--- Up24.dat ---
&ACCESS RVO1
&REL 1255
&COMMENT VW380 Klebeauftrag_AFO415600
&PARAM EDITMASK = Up999[1-999]
&PARAM TEMPLATE = C:\KRC\Roboter\Template\upvorgabe
&PARAM TPVW_VERSION = 8.3.18
&PARAM DISKPATH = KRC:\R1\UPs
DEFDAT UP24
; FOLD ;%{H} %MKUKATPVW
; ENDFOLD
; interface to basic routines
 EXT  BAS (BAS_COMMAND  :IN,REAL  :IN )
; interface to VW-standard routines
EXT VW (VW_COMMAND:IN, BOOL: IN, REAL:IN, REAL:IN, REAL:IN, REAL:IN, BOOL :IN, E6POS :IN )
; interface to VW_USER - Call
EXT  VW_USER (VW_USER_CMD :IN,INT :IN,REAL  :IN,REAL  :IN,REAL  :IN,REAL  :IN,REAL  :IN,REAL  :IN,REAL  :IN,REAL  :IN,REAL  :IN,BOOL  :IN)
EXT  VW_USR_R (VW_USER_CMD :IN,INT :IN,REAL  :IN,REAL  :IN,REAL  :IN,REAL  :IN,REAL  :IN,REAL  :IN,REAL  :IN,REAL  :IN,REAL  :IN,BOOL  :IN)
EXT  IBGN (IBGN_COMMAND  :IN,BOOL  :IN,REAL  :IN,REAL  :IN,BOOL  :IN,E6POS  :OUT )
; interface select routine
EXTFCT INT  SELECT (SUBTYPE  :IN,INT  :IN,BOOL  :IN,ARI_TYP  :IN,INT  :IN,BOOL_TYP  :IN,INT  :IN,BOOL  :IN)
INT VW_NEXT_FREE = 145
INT VW_NFREE_SPS = 147
INT VW_MAX_SPS = 247
DECL VW_MPARA_TYP P1_D = {TOOL_NO 1,BASE_NO 2,VB 100,VE 0,ACC 100,TRG_TIME 0,MOVE_TYPE #PTP_MOTION}
DECL E6POS P1 = {X 1079.993, Y 23.2307, Z -59.63425, A -156.517, B 2.823335, C 116.2772, S 2, T 2 , E1 0.0, E2 0.0, E3 0.0, E4 0.0, E5 0.0, E6 0.0}
DECL VW_MPARA_TYP P2_D = {TOOL_NO 1,BASE_NO 2,VB 100,VE 100,ACC 100,TRG_TIME 0,MOVE_TYPE #PTP_MOTION}
DECL E6POS P2 = {X 1309.031, Y -94.76365, Z 183.6622, A -143.6638, B -5.59984, C 155.4084, S 2, T 2 , E1 0.0, E2 0.0, E3 0.0, E4 0.0, E5 0.0, E6 0.0}
DECL VW_MPARA_TYP P3_D = {TOOL_NO 1,BASE_NO 2,VB 100,VE 100,ACC 100,TRG_TIME 0,MOVE_TYPE #PTP_MOTION}
DECL E6POS P3 = {X 2315.081, Y -270.0302, Z 820.4095, A -112.6535, B -26.53998, C -109.4264, S 2, T 34 , E1 0.0, E2 0.0, E3 0.0, E4 0.0, E5 0.0, E6 0.0}
DECL VW_MPARA_TYP P4_D = {TOOL_NO 1,BASE_NO 2,VB 100,VE 100,ACC 100,TRG_TIME 0,MOVE_TYPE #PTP_MOTION}
DECL E6POS P4 = {X 2638.59, Y -718.27, Z 643.3, A -85.45, B -17.603, C 1.681, S 2, T 34 , E1 0.0, E2 0.0, E3 0.0, E4 0.0, E5 0.0, E6 0.0}
DECL VW_MPARA_TYP P5_D = {TOOL_NO 1,BASE_NO 2,VB 100,VE 0,ACC 100,TRG_TIME 0,MOVE_TYPE #PTP_MOTION}
DECL E6POS P5 = {X 2551.881, Y -682.7541, Z 739.713, A -85.45, B -17.603, C 36.73906, S 2, T 34 , E1 0.0, E2 0.0, E3 0.0, E4 0.0, E5 0.0, E6 0.0}
DECL VW_MPARA_TYP P6_D = {TOOL_NO 1,BASE_NO 2,VB 150,VE 30,ACC 50,TRG_TIME 0,MOVE_TYPE #GLUE_MOTION}
DECL E6POS P6 = {X 2504.219, Y -701.0809, Z 748.469, A -85.45, B -17.603, C 40.17007, S 2, T 34 , E1 0.0, E2 0.0, E3 0.0, E4 0.0, E5 0.0, E6 0.0}
DECL VW_MPARA_TYP P7_D = {TOOL_NO 1,BASE_NO 2,VB 150,VE 30,ACC 50,TRG_TIME 5,MOVE_TYPE #GLUE_MOTION}
DECL E6POS P7 = {X 2478.381, Y -706.9081, Z 747.4919, A -85.45, B -17.603, C 40.17007, S 2, T 34 , E1 0.0, E2 0.0, E3 0.0, E4 0.0, E5 0.0, E6 0.0}
DECL VW_MPARA_TYP P8_D = {TOOL_NO 1,BASE_NO 2,VB 150,VE 30,ACC 50,TRG_TIME 5,MOVE_TYPE #GLUE_MOTION}
DECL E6POS P8 = {X 2410.503, Y -712.4858, Z 745.5424, A -85.83325, B -17.36149, C 46.89683, S 2, T 34 , E1 0.0, E2 0.0, E3 0.0, E4 0.0, E5 0.0, E6 0.0}
DECL VW_MPARA_TYP P9_D = {TOOL_NO 1,BASE_NO 2,VB 150,VE 30,ACC 50,TRG_TIME 0,MOVE_TYPE #GLUE_MOTION}
DECL E6POS P9 = {X 2390.268, Y -711.3152, Z 744.5164, A -85.94926, B -17.28811, C 48.93612, S 2, T 34 , E1 0.0, E2 0.0, E3 0.0, E4 0.0, E5 0.0, E6 0.0}
DECL VW_MPARA_TYP P10_D = {TOOL_NO 1,BASE_NO 2,VB 200,VE 40,ACC 50,TRG_TIME 0,MOVE_TYPE #GLUE_MOTION}
DECL E6POS P10 = {X 2368.57, Y -713.33, Z 742.9525, A -86.064, B -17.2163, C 50.87427, S 2, T 34 , E1 0.0, E2 0.0, E3 0.0, E4 0.0, E5 0.0, E6 0.0}
DECL VW_MPARA_TYP P11_D = {TOOL_NO 1,BASE_NO 2,VB 200,VE 40,ACC 50,TRG_TIME 5,MOVE_TYPE #GLUE_MOTION}
DECL E6POS P11 = {X 2345.222, Y -717.935, Z 743.7926, A -86.1802, B -17.14345, C 52.83833, S 2, T 34 , E1 0.0, E2 0.0, E3 0.0, E4 0.0, E5 0.0, E6 0.0}
DECL VW_MPARA_TYP P12_D = {TOOL_NO 1,BASE_NO 2,VB 200,VE 40,ACC 50,TRG_TIME 0,MOVE_TYPE #GLUE_MOTION}
DECL E6POS P12 = {X 2323.359, Y -720.4127, Z 742.2736, A -86.30313, B -17.06625, C 54.91773, S 2, T 34 , E1 0.0, E2 0.0, E3 0.0, E4 0.0, E5 0.0, E6 0.0}
DECL VW_MPARA_TYP P13_D = {TOOL_NO 1,BASE_NO 2,VB 200,VE 40,ACC 50,TRG_TIME 5,MOVE_TYPE #GLUE_MOTION}
DECL E6POS P13 = {X 2240.693, Y -726.2643, Z 739.3849, A -86.74549, B -16.78729, C 62.41298, S 2, T 42 , E1 0.0, E2 0.0, E3 0.0, E4 0.0, E5 0.0, E6 0.0}
DECL VW_MPARA_TYP P14_D = {TOOL_NO 1,BASE_NO 2,VB 200,VE 40,ACC 50,TRG_TIME 0,MOVE_TYPE #GLUE_MOTION}
DECL E6POS P14 = {X 2221.286, Y -727.9705, Z 739.491, A -86.84053, B -16.72713, C 64.02588, S 2, T 42 , E1 0.0, E2 0.0, E3 0.0, E4 0.0, E5 0.0, E6 0.0}
DECL VW_MPARA_TYP P15_D = {TOOL_NO 1,BASE_NO 2,VB 200,VE 40,ACC 50,TRG_TIME 0,MOVE_TYPE #GLUE_MOTION}
DECL E6POS P15 = {X 2177.699, Y -731.3578, Z 738.373, A -86.928, B -16.688, C 64.0209, S 2, T 42 , E1 0.0, E2 0.0, E3 0.0, E4 0.0, E5 0.0, E6 0.0}
DECL VW_MPARA_TYP P16_D = {TOOL_NO 1,BASE_NO 2,VB 200,VE 40,ACC 50,TRG_TIME 0,MOVE_TYPE #GLUE_MOTION}
DECL E6POS P16 = {X 2146.549, Y -733.2928, Z 737.3707, A -86.99107, B -16.6619, C 64.0342, S 2, T 42 , E1 0.0, E2 0.0, E3 0.0, E4 0.0, E5 0.0, E6 0.0}
DECL VW_MPARA_TYP P17_D = {TOOL_NO 1,BASE_NO 2,VB 200,VE 40,ACC 50,TRG_TIME 0,MOVE_TYPE #GLUE_MOTION}
DECL E6POS P17 = {X 2071.937, Y -738.6399, Z 734.6805, A -87.14213, B -16.59928, C 64.02824, S 2, T 42 , E1 0.0, E2 0.0, E3 0.0, E4 0.0, E5 0.0, E6 0.0}
DECL VW_MPARA_TYP P18_D = {TOOL_NO 1,BASE_NO 2,VB 200,VE 40,ACC 50,TRG_TIME 0,MOVE_TYPE #GLUE_MOTION}
DECL E6POS P18 = {X 1997.84, Y -742.9333, Z 732.2686, A -87.292, B -16.537, C 64.03024, S 2, T 42 , E1 0.0, E2 0.0, E3 0.0, E4 0.0, E5 0.0, E6 0.0}
DECL VW_MPARA_TYP P19_D = {TOOL_NO 1,BASE_NO 2,VB 200,VE 40,ACC 50,TRG_TIME 0,MOVE_TYPE #GLUE_MOTION}
DECL E6POS P19 = {X 1957.689, Y -745.717, Z 730.7956, A -87.3728, B -16.5027, C 64.02561, S 2, T 42 , E1 0.0, E2 0.0, E3 0.0, E4 0.0, E5 0.0, E6 0.0}
DECL VW_MPARA_TYP P20_D = {TOOL_NO 1,BASE_NO 2,VB 200,VE 40,ACC 50,TRG_TIME 0,MOVE_TYPE #GLUE_MOTION}
DECL E6POS P20 = {X 1924.073, Y -747.3588, Z 729.5613, A -87.44041, B -16.47397, C 64.02909, S 2, T 42 , E1 0.0, E2 0.0, E3 0.0, E4 0.0, E5 0.0, E6 0.0}
DECL VW_MPARA_TYP P21_D = {TOOL_NO 1,BASE_NO 2,VB 200,VE 40,ACC 50,TRG_TIME 0,MOVE_TYPE #GLUE_MOTION}
DECL E6POS P21 = {X 1839.674, Y -751.9378, Z 726.4262, A -87.6101, B -16.40172, C 64.02763, S 2, T 42 , E1 0.0, E2 0.0, E3 0.0, E4 0.0, E5 0.0, E6 0.0}
DECL VW_MPARA_TYP P22_D = {TOOL_NO 1,BASE_NO 2,VB 200,VE 40,ACC 50,TRG_TIME 0,MOVE_TYPE #GLUE_MOTION}
DECL E6POS P22 = {X 1817.83, Y -753.1229, Z 725.5301, A -87.654, B -16.383, C 64.02721, S 2, T 42 , E1 0.0, E2 0.0, E3 0.0, E4 0.0, E5 0.0, E6 0.0}
DECL VW_MPARA_TYP P23_D = {TOOL_NO 1,BASE_NO 2,VB 200,VE 40,ACC 50,TRG_TIME 0,MOVE_TYPE #GLUE_MOTION}
DECL E6POS P23 = {X 1809.814, Y -753.5765, Z 724.9373, A -87.68093, B -16.37124, C 64.02778, S 2, T 42 , E1 0.0, E2 0.0, E3 0.0, E4 0.0, E5 0.0, E6 0.0}
DECL VW_MPARA_TYP P24_D = {TOOL_NO 1,BASE_NO 2,VB 200,VE 40,ACC 50,TRG_TIME 0,MOVE_TYPE #GLUE_MOTION}
DECL E6POS P24 = {X 1802.477, Y -755.0577, Z 721.8582, A -87.69443, B -16.36536, C 64.02803, S 2, T 42 , E1 0.0, E2 0.0, E3 0.0, E4 0.0, E5 0.0, E6 0.0}
DECL VW_MPARA_TYP P25_D = {TOOL_NO 1,BASE_NO 2,VB 200,VE 40,ACC 50,TRG_TIME 0,MOVE_TYPE #GLUE_MOTION}
DECL E6POS P25 = {X 1798.327, Y -755.0577, Z 721.8582, A -87.69443, B -16.36536, C 64.02803, S 2, T 42 , E1 0.0, E2 0.0, E3 0.0, E4 0.0, E5 0.0, E6 0.0}
DECL VW_MPARA_TYP P26_D = {TOOL_NO 1,BASE_NO 2,VB 200,VE 40,ACC 50,TRG_TIME 0,MOVE_TYPE #GLUE_MOTION}
DECL E6POS P26 = {X 1789.116, Y -754.8168, Z 723.4621, A -87.71136, B -16.35797, C 64.02837, S 2, T 42 , E1 0.0, E2 0.0, E3 0.0, E4 0.0, E5 0.0, E6 0.0}
DECL VW_MPARA_TYP P27_D = {TOOL_NO 1,BASE_NO 2,VB 200,VE 40,ACC 50,TRG_TIME 0,MOVE_TYPE #GLUE_MOTION}
DECL E6POS P27 = {X 1750.697, Y -755.6901, Z 722.3646, A -87.79472, B -16.32156, C 64.03, S 2, T 42 , E1 0.0, E2 0.0, E3 0.0, E4 0.0, E5 0.0, E6 0.0}
DECL VW_MPARA_TYP P28_D = {TOOL_NO 1,BASE_NO 2,VB 200,VE 40,ACC 50,TRG_TIME 0,MOVE_TYPE #GLUE_MOTION}
DECL E6POS P28 = {X 1688.285, Y -758.5743, Z 719.4387, A -87.92546, B -16.26436, C 64.03244, S 2, T 42 , E1 0.0, E2 0.0, E3 0.0, E4 0.0, E5 0.0, E6 0.0}
DECL VW_MPARA_TYP P29_D = {TOOL_NO 1,BASE_NO 2,VB 200,VE 40,ACC 50,TRG_TIME 5,MOVE_TYPE #GLUE_MOTION}
DECL E6POS P29 = {X 1641.474, Y -760.4988, Z 718.2494, A -88.013, B -16.226, C 64.03399, S 2, T 42 , E1 0.0, E2 0.0, E3 0.0, E4 0.0, E5 0.0, E6 0.0}
DECL VW_MPARA_TYP P30_D = {TOOL_NO 1,BASE_NO 2,VB 200,VE 40,ACC 50,TRG_TIME 0,MOVE_TYPE #GLUE_MOTION}
DECL E6POS P30 = {X 1627.713, Y -759.5684, Z 718.5726, A -88.013, B -16.22599, C 64.02855, S 2, T 42 , E1 0.0, E2 0.0, E3 0.0, E4 0.0, E5 0.0, E6 0.0}
DECL VW_MPARA_TYP P31_D = {TOOL_NO 1,BASE_NO 2,VB 150,VE 30,ACC 50,TRG_TIME 0,MOVE_TYPE #GLUE_MOTION}
DECL E6POS P31 = {X 1593.2, Y -759.0589, Z 716.3181, A -88.013, B -16.226, C 64.03667, S 2, T 42 , E1 0.0, E2 0.0, E3 0.0, E4 0.0, E5 0.0, E6 0.0}
DECL VW_MPARA_TYP P32_D = {TOOL_NO 1,BASE_NO 2,VB 150,VE 30,ACC 50,TRG_TIME 5,MOVE_TYPE #GLUE_MOTION}
DECL E6POS P32 = {X 1572.434, Y -763.546, Z 715.0018, A -88.986, B -15.66601, C 64.04243, S 2, T 42 , E1 0.0, E2 0.0, E3 0.0, E4 0.0, E5 0.0, E6 0.0}
DECL VW_MPARA_TYP P33_D = {TOOL_NO 1,BASE_NO 2,VB 150,VE 30,ACC 50,TRG_TIME 0,MOVE_TYPE #GLUE_MOTION}
DECL E6POS P33 = {X 1555.049, Y -763.8819, Z 714.8086, A -88.986, B -15.66601, C 64.02816, S 2, T 42 , E1 0.0, E2 0.0, E3 0.0, E4 0.0, E5 0.0, E6 0.0}
DECL VW_MPARA_TYP P34_D = {TOOL_NO 1,BASE_NO 2,VB 150,VE 30,ACC 50,TRG_TIME 5,MOVE_TYPE #GLUE_MOTION}
DECL E6POS P34 = {X 1524.233, Y -764.9556, Z 712.8458, A -88.986, B -15.666, C 64.02997, S 2, T 42 , E1 0.0, E2 0.0, E3 0.0, E4 0.0, E5 0.0, E6 0.0}
DECL VW_MPARA_TYP P35_D = {TOOL_NO 1,BASE_NO 2,VB 150,VE 30,ACC 50,TRG_TIME 0,MOVE_TYPE #GLUE_MOTION}
DECL E6POS P35 = {X 1511.87, Y -762.7119, Z 711.4664, A -88.986, B -15.666, C 64.02997, S 2, T 42 , E1 0.0, E2 0.0, E3 0.0, E4 0.0, E5 0.0, E6 0.0}
DECL VW_MPARA_TYP P36_D = {TOOL_NO 1,BASE_NO 2,VB 300,VE 10,ACC 50,TRG_TIME 0,MOVE_TYPE #PATH_MOTION}
DECL E6POS P36 = {X 1503.42, Y -769.8487, Z 701.9658, A -88.07185, B -1.118032, C 83.01237, S 2, T 42 , E1 0.0, E2 0.0, E3 0.0, E4 0.0, E5 0.0, E6 0.0}
DECL VW_MPARA_TYP P37_D = {TOOL_NO 1,BASE_NO 2,VB 200,VE 40,ACC 50,TRG_TIME 0,MOVE_TYPE #GLUE_MOTION}
DECL E6POS P37 = {X 1503.42, Y -769.8487, Z 697.7132, A -88.07185, B -1.118032, C 83.01237, S 2, T 42 , E1 0.0, E2 0.0, E3 0.0, E4 0.0, E5 0.0, E6 0.0}
DECL VW_MPARA_TYP P38_D = {TOOL_NO 1,BASE_NO 2,VB 200,VE 40,ACC 50,TRG_TIME 5,MOVE_TYPE #GLUE_MOTION}
DECL E6POS P38 = {X 1499.395, Y -778.1977, Z 683.0693, A -88.07185, B -1.118032, C 83.01237, S 2, T 42 , E1 0.0, E2 0.0, E3 0.0, E4 0.0, E5 0.0, E6 0.0}
DECL VW_MPARA_TYP P39_D = {TOOL_NO 1,BASE_NO 2,VB 200,VE 40,ACC 50,TRG_TIME 0,MOVE_TYPE #GLUE_MOTION}
DECL E6POS P39 = {X 1498.217, Y -783.5937, Z 672.2539, A -88.04707, B -1.074359, C 83.00169, S 2, T 42 , E1 0.0, E2 0.0, E3 0.0, E4 0.0, E5 0.0, E6 0.0}
DECL VW_MPARA_TYP P40_D = {TOOL_NO 1,BASE_NO 2,VB 200,VE 40,ACC 50,TRG_TIME 0,MOVE_TYPE #GLUE_MOTION}
DECL E6POS P40 = {X 1493.03, Y -794.5521, Z 652.6918, A -88.02206, B -1.060599, C 83.00537, S 2, T 42 , E1 0.0, E2 0.0, E3 0.0, E4 0.0, E5 0.0, E6 0.0}
DECL VW_MPARA_TYP P41_D = {TOOL_NO 1,BASE_NO 2,VB 200,VE 40,ACC 50,TRG_TIME 0,MOVE_TYPE #GLUE_MOTION}
DECL E6POS P41 = {X 1488.754, Y -807.0863, Z 632.17, A -88.03383, B -1.06127, C 83.01902, S 2, T 42 , E1 0.0, E2 0.0, E3 0.0, E4 0.0, E5 0.0, E6 0.0}
DECL VW_MPARA_TYP P42_D = {TOOL_NO 1,BASE_NO 2,VB 200,VE 40,ACC 50,TRG_TIME 0,MOVE_TYPE #GLUE_MOTION}
DECL E6POS P42 = {X 1485.688, Y -814.9008, Z 620.4972, A -88.01247, B -0.993889, C 82.99284, S 2, T 42 , E1 0.0, E2 0.0, E3 0.0, E4 0.0, E5 0.0, E6 0.0}
DECL VW_MPARA_TYP P43_D = {TOOL_NO 1,BASE_NO 2,VB 200,VE 40,ACC 50,TRG_TIME 0,MOVE_TYPE #GLUE_MOTION}
DECL E6POS P43 = {X 1481.476, Y -827.8041, Z 605.2604, A -88.01193, B -0.994103, C 83.00861, S 2, T 42 , E1 0.0, E2 0.0, E3 0.0, E4 0.0, E5 0.0, E6 0.0}
DECL VW_MPARA_TYP P44_D = {TOOL_NO 1,BASE_NO 2,VB 200,VE 40,ACC 50,TRG_TIME 0,MOVE_TYPE #GLUE_MOTION}
DECL E6POS P44 = {X 1478.198, Y -834.6122, Z 593.0376, A -88.05488, B 1.000137, C 83.08899, S 2, T 42 , E1 0.0, E2 0.0, E3 0.0, E4 0.0, E5 0.0, E6 0.0}
DECL VW_MPARA_TYP P45_D = {TOOL_NO 1,BASE_NO 2,VB 200,VE 40,ACC 50,TRG_TIME 0,MOVE_TYPE #GLUE_MOTION}
DECL E6POS P45 = {X 1476.832, Y -836.955, Z 579.7414, A -88.0008, B 0.989837, C 83.0631, S 2, T 42 , E1 0.0, E2 0.0, E3 0.0, E4 0.0, E5 0.0, E6 0.0}
DECL VW_MPARA_TYP P46_D = {TOOL_NO 1,BASE_NO 2,VB 200,VE 40,ACC 50,TRG_TIME 0,MOVE_TYPE #GLUE_MOTION}
DECL E6POS P46 = {X 1473.648, Y -841.1156, Z 561.5488, A -88.05322, B 1.024646, C 83.01369, S 2, T 42 , E1 0.0, E2 0.0, E3 0.0, E4 0.0, E5 0.0, E6 0.0}
DECL VW_MPARA_TYP P47_D = {TOOL_NO 1,BASE_NO 2,VB 200,VE 40,ACC 50,TRG_TIME 0,MOVE_TYPE #GLUE_MOTION}
DECL E6POS P47 = {X 1471.16, Y -846.8204, Z 536.7025, A -87.97337, B 0.987811, C 83.00545, S 2, T 42 , E1 0.0, E2 0.0, E3 0.0, E4 0.0, E5 0.0, E6 0.0}
DECL VW_MPARA_TYP P48_D = {TOOL_NO 1,BASE_NO 2,VB 200,VE 40,ACC 50,TRG_TIME 0,MOVE_TYPE #GLUE_MOTION}
DECL E6POS P48 = {X 1465.512, Y -853.3635, Z 505.8478, A -88.0125, B 1.009102, C 83.03255, S 2, T 42 , E1 0.0, E2 0.0, E3 0.0, E4 0.0, E5 0.0, E6 0.0}
DECL VW_MPARA_TYP P49_D = {TOOL_NO 1,BASE_NO 2,VB 200,VE 40,ACC 50,TRG_TIME 0,MOVE_TYPE #GLUE_MOTION}
DECL E6POS P49 = {X 1463.656, Y -855.4403, Z 486.6357, A -88.05423, B 1.001739, C 82.99404, S 2, T 42 , E1 0.0, E2 0.0, E3 0.0, E4 0.0, E5 0.0, E6 0.0}
DECL VW_MPARA_TYP P50_D = {TOOL_NO 1,BASE_NO 2,VB 200,VE 40,ACC 50,TRG_TIME 0,MOVE_TYPE #GLUE_MOTION}
DECL E6POS P50 = {X 1461.566, Y -857.1955, Z 468.6439, A -88.00505, B 1.002154, C 83.01239, S 2, T 42 , E1 0.0, E2 0.0, E3 0.0, E4 0.0, E5 0.0, E6 0.0}
DECL VW_MPARA_TYP P51_D = {TOOL_NO 1,BASE_NO 2,VB 200,VE 40,ACC 50,TRG_TIME 0,MOVE_TYPE #GLUE_MOTION}
DECL E6POS P51 = {X 1458.06, Y -858.806, Z 451.0082, A -88.02662, B 1.033577, C 83.00974, S 2, T 42 , E1 0.0, E2 0.0, E3 0.0, E4 0.0, E5 0.0, E6 0.0}
DECL VW_MPARA_TYP P52_D = {TOOL_NO 1,BASE_NO 2,VB 200,VE 40,ACC 50,TRG_TIME 0,MOVE_TYPE #GLUE_MOTION}
DECL E6POS P52 = {X 1457.169, Y -859.5342, Z 426.4188, A -88.01513, B 1.012713, C 83.00486, S 2, T 42 , E1 0.0, E2 0.0, E3 0.0, E4 0.0, E5 0.0, E6 0.0}
DECL VW_MPARA_TYP P53_D = {TOOL_NO 1,BASE_NO 2,VB 200,VE 40,ACC 50,TRG_TIME 0,MOVE_TYPE #GLUE_MOTION}
DECL E6POS P53 = {X 1457.207, Y -860.6595, Z 406.3141, A -88.02609, B 1.004751, C 83.00697, S 2, T 42 , E1 0.0, E2 0.0, E3 0.0, E4 0.0, E5 0.0, E6 0.0}
DECL VW_MPARA_TYP P54_D = {TOOL_NO 1,BASE_NO 2,VB 200,VE 40,ACC 50,TRG_TIME 0,MOVE_TYPE #GLUE_MOTION}
DECL E6POS P54 = {X 1455.6, Y -859.7858, Z 384.9504, A -88.00213, B 1.035148, C 83.0168, S 2, T 42 , E1 0.0, E2 0.0, E3 0.0, E4 0.0, E5 0.0, E6 0.0}
DECL VW_MPARA_TYP P55_D = {TOOL_NO 1,BASE_NO 2,VB 200,VE 40,ACC 50,TRG_TIME 0,MOVE_TYPE #GLUE_MOTION}
DECL E6POS P55 = {X 1455.86, Y -859.1099, Z 365.5491, A -87.99634, B 1.010499, C 83.00358, S 2, T 42 , E1 0.0, E2 0.0, E3 0.0, E4 0.0, E5 0.0, E6 0.0}
DECL VW_MPARA_TYP P56_D = {TOOL_NO 1,BASE_NO 2,VB 200,VE 40,ACC 50,TRG_TIME 0,MOVE_TYPE #GLUE_MOTION}
DECL E6POS P56 = {X 1454.703, Y -858.3672, Z 343.593, A -88.00025, B 0.997425, C 82.98918, S 2, T 42 , E1 0.0, E2 0.0, E3 0.0, E4 0.0, E5 0.0, E6 0.0}
DECL VW_MPARA_TYP P57_D = {TOOL_NO 1,BASE_NO 2,VB 200,VE 40,ACC 50,TRG_TIME 0,MOVE_TYPE #GLUE_MOTION}
DECL E6POS P57 = {X 1453.179, Y -857.4509, Z 316.5913, A -87.99828, B 1.004134, C 83.0314, S 2, T 42 , E1 0.0, E2 0.0, E3 0.0, E4 0.0, E5 0.0, E6 0.0}
DECL VW_MPARA_TYP P58_D = {TOOL_NO 1,BASE_NO 2,VB 200,VE 40,ACC 50,TRG_TIME 0,MOVE_TYPE #GLUE_MOTION}
DECL E6POS P58 = {X 1452.497, Y -854.6255, Z 291.8859, A -88.00141, B 1.058003, C 82.99638, S 2, T 42 , E1 0.0, E2 0.0, E3 0.0, E4 0.0, E5 0.0, E6 0.0}
DECL VW_MPARA_TYP P59_D = {TOOL_NO 1,BASE_NO 2,VB 200,VE 40,ACC 50,TRG_TIME 0,MOVE_TYPE #GLUE_MOTION}
DECL E6POS P59 = {X 1451.678, Y -852.0793, Z 264.5305, A -88.0264, B 0.995717, C 83.0143, S 2, T 42 , E1 0.0, E2 0.0, E3 0.0, E4 0.0, E5 0.0, E6 0.0}
DECL VW_MPARA_TYP P60_D = {TOOL_NO 1,BASE_NO 2,VB 200,VE 40,ACC 50,TRG_TIME 0,MOVE_TYPE #GLUE_MOTION}
DECL E6POS P60 = {X 1451.391, Y -849.9799, Z 239.6057, A -88.01192, B 0.999021, C 82.99754, S 2, T 42 , E1 0.0, E2 0.0, E3 0.0, E4 0.0, E5 0.0, E6 0.0}
DECL VW_MPARA_TYP P61_D = {TOOL_NO 1,BASE_NO 2,VB 200,VE 40,ACC 50,TRG_TIME 0,MOVE_TYPE #GLUE_MOTION}
DECL E6POS P61 = {X 1452.496, Y -848.1734, Z 217.2187, A -88.01024, B 1.007652, C 83.08875, S 2, T 42 , E1 0.0, E2 0.0, E3 0.0, E4 0.0, E5 0.0, E6 0.0}
DECL VW_MPARA_TYP P62_D = {TOOL_NO 1,BASE_NO 2,VB 200,VE 40,ACC 50,TRG_TIME 0,MOVE_TYPE #GLUE_MOTION}
DECL E6POS P62 = {X 1452.505, Y -846.1744, Z 193.6873, A -88.03108, B 1.004962, C 82.99518, S 2, T 42 , E1 0.0, E2 0.0, E3 0.0, E4 0.0, E5 0.0, E6 0.0}
DECL VW_MPARA_TYP P63_D = {TOOL_NO 1,BASE_NO 2,VB 200,VE 40,ACC 50,TRG_TIME 0,MOVE_TYPE #GLUE_MOTION}
DECL E6POS P63 = {X 1452.866, Y -848.0626, Z 170.8705, A -88.01171, B 1.00305, C 83.03461, S 2, T 42 , E1 0.0, E2 0.0, E3 0.0, E4 0.0, E5 0.0, E6 0.0}
DECL VW_MPARA_TYP P64_D = {TOOL_NO 1,BASE_NO 2,VB 200,VE 40,ACC 50,TRG_TIME 0,MOVE_TYPE #GLUE_MOTION}
DECL E6POS P64 = {X 1454.113, Y -850.143, Z 146.9456, A -87.99117, B 1.002189, C 82.9839, S 2, T 42 , E1 0.0, E2 0.0, E3 0.0, E4 0.0, E5 0.0, E6 0.0}
DECL VW_MPARA_TYP P65_D = {TOOL_NO 1,BASE_NO 2,VB 200,VE 40,ACC 50,TRG_TIME 0,MOVE_TYPE #GLUE_MOTION}
DECL E6POS P65 = {X 1454.352, Y -851.0382, Z 135.797, A -88.0205, B 1.002176, C 82.99446, S 2, T 42 , E1 0.0, E2 0.0, E3 0.0, E4 0.0, E5 0.0, E6 0.0}
DECL VW_MPARA_TYP P66_D = {TOOL_NO 1,BASE_NO 2,VB 200,VE 40,ACC 50,TRG_TIME 0,MOVE_TYPE #GLUE_MOTION}
DECL E6POS P66 = {X 1455.34, Y -852.0748, Z 122.3131, A -87.99885, B 0.987187, C 83.00255, S 2, T 42 , E1 0.0, E2 0.0, E3 0.0, E4 0.0, E5 0.0, E6 0.0}
DECL VW_MPARA_TYP P67_D = {TOOL_NO 1,BASE_NO 2,VB 200,VE 40,ACC 50,TRG_TIME 0,MOVE_TYPE #GLUE_MOTION}
DECL E6POS P67 = {X 1455.695, Y -853.7063, Z 108.5957, A -87.99349, B 1.005062, C 83.07543, S 2, T 42 , E1 0.0, E2 0.0, E3 0.0, E4 0.0, E5 0.0, E6 0.0}
DECL VW_MPARA_TYP P68_D = {TOOL_NO 1,BASE_NO 2,VB 200,VE 40,ACC 50,TRG_TIME 0,MOVE_TYPE #GLUE_MOTION}
DECL E6POS P68 = {X 1456.311, Y -854.9208, Z 97.20465, A -88.00738, B 1.004484, C 82.99986, S 2, T 42 , E1 0.0, E2 0.0, E3 0.0, E4 0.0, E5 0.0, E6 0.0}
DECL VW_MPARA_TYP P69_D = {TOOL_NO 1,BASE_NO 2,VB 200,VE 40,ACC 50,TRG_TIME 0,MOVE_TYPE #GLUE_MOTION}
DECL E6POS P69 = {X 1457.166, Y -854.1422, Z 84.21948, A -88.01357, B 1.019535, C 82.99683, S 2, T 42 , E1 0.0, E2 0.0, E3 0.0, E4 0.0, E5 0.0, E6 0.0}
DECL VW_MPARA_TYP P70_D = {TOOL_NO 1,BASE_NO 2,VB 200,VE 40,ACC 50,TRG_TIME 0,MOVE_TYPE #GLUE_MOTION}
DECL E6POS P70 = {X 1459.489, Y -851.3946, Z 71.32433, A -88.01587, B 1.021121, C 82.9754, S 2, T 42 , E1 0.0, E2 0.0, E3 0.0, E4 0.0, E5 0.0, E6 0.0}
DECL VW_MPARA_TYP P71_D = {TOOL_NO 1,BASE_NO 2,VB 200,VE 40,ACC 50,TRG_TIME 0,MOVE_TYPE #GLUE_MOTION}
DECL E6POS P71 = {X 1460.998, Y -847.6905, Z 60.30585, A -87.9896, B 1.003461, C 82.99796, S 2, T 42 , E1 0.0, E2 0.0, E3 0.0, E4 0.0, E5 0.0, E6 0.0}
DECL VW_MPARA_TYP P72_D = {TOOL_NO 1,BASE_NO 2,VB 200,VE 40,ACC 50,TRG_TIME 5,MOVE_TYPE #GLUE_MOTION}
DECL E6POS P72 = {X 1460.858, Y -845.861, Z 56.39811, A -88.006, B 1.00273, C 83.00398, S 2, T 42 , E1 0.0, E2 0.0, E3 0.0, E4 0.0, E5 0.0, E6 0.0}
DECL VW_MPARA_TYP P73_D = {TOOL_NO 1,BASE_NO 2,VB 200,VE 40,ACC 50,TRG_TIME 0,MOVE_TYPE #GLUE_MOTION}
DECL E6POS P73 = {X 1465.282, Y -838.3979, Z 33.94293, A -87.996, B 0.996512, C 82.99879, S 2, T 42 , E1 0.0, E2 0.0, E3 0.0, E4 0.0, E5 0.0, E6 0.0}
DECL VW_MPARA_TYP P74_D = {TOOL_NO 1,BASE_NO 2,VB 100,VE 100,ACC 100,TRG_TIME 0,MOVE_TYPE #PTP_MOTION}
DECL E6POS P74 = {X 1476.75, Y -808.8141, Z 29.90171, A -87.314, B 15.48001, C 64.62599, S 2, T 34 , E1 0.0, E2 0.0, E3 0.0, E4 0.0, E5 0.0, E6 0.0}
DECL VW_MPARA_TYP P75_D = {TOOL_NO 1,BASE_NO 2,VB 100,VE 100,ACC 100,TRG_TIME 0,MOVE_TYPE #PTP_MOTION}
DECL E6POS P75 = {X 1491.529, Y -835.7732, Z 79.1761, A -87.98852, B 16.99558, C 60.00438, S 2, T 34 , E1 0.0, E2 0.0, E3 0.0, E4 0.0, E5 0.0, E6 0.0}
DECL VW_MPARA_TYP P76_D = {TOOL_NO 1,BASE_NO 2,VB 200,VE 40,ACC 50,TRG_TIME 0,MOVE_TYPE #GLUE_MOTION}
DECL E6POS P76 = {X 1476.06, Y -853.2753, Z 52.70673, A -87.98852, B 16.99558, C 60.00438, S 2, T 34 , E1 0.0, E2 0.0, E3 0.0, E4 0.0, E5 0.0, E6 0.0}
DECL VW_MPARA_TYP P77_D = {TOOL_NO 1,BASE_NO 2,VB 200,VE 40,ACC 50,TRG_TIME 5,MOVE_TYPE #GLUE_MOTION}
DECL E6POS P77 = {X 1475.091, Y -849.7084, Z 38.60646, A -87.98852, B 16.99558, C 60.00438, S 2, T 34 , E1 0.0, E2 0.0, E3 0.0, E4 0.0, E5 0.0, E6 0.0}
DECL VW_MPARA_TYP P78_D = {TOOL_NO 1,BASE_NO 2,VB 200,VE 40,ACC 50,TRG_TIME 0,MOVE_TYPE #GLUE_MOTION}
DECL E6POS P78 = {X 1480.383, Y -846.2617, Z 27.19039, A -88.00126, B 17.00734, C 59.98072, S 2, T 34 , E1 0.0, E2 0.0, E3 0.0, E4 0.0, E5 0.0, E6 0.0}
DECL VW_MPARA_TYP P79_D = {TOOL_NO 1,BASE_NO 2,VB 200,VE 40,ACC 50,TRG_TIME 0,MOVE_TYPE #GLUE_MOTION}
DECL E6POS P79 = {X 1529.002, Y -845.3863, Z 29.04734, A -88.05003, B 17.03112, C 60.00431, S 2, T 34 , E1 0.0, E2 0.0, E3 0.0, E4 0.0, E5 0.0, E6 0.0}
DECL VW_MPARA_TYP P80_D = {TOOL_NO 1,BASE_NO 2,VB 200,VE 40,ACC 50,TRG_TIME 0,MOVE_TYPE #GLUE_MOTION}
DECL E6POS P80 = {X 1548.778, Y -845.3863, Z 30.24737, A -88.05003, B 17.03112, C 60.00431, S 2, T 34 , E1 0.0, E2 0.0, E3 0.0, E4 0.0, E5 0.0, E6 0.0}
DECL VW_MPARA_TYP P81_D = {TOOL_NO 1,BASE_NO 2,VB 200,VE 40,ACC 50,TRG_TIME 0,MOVE_TYPE #GLUE_MOTION}
DECL E6POS P81 = {X 1590.973, Y -844.937, Z 34.43459, A -88.00398, B 17.00217, C 60.00132, S 2, T 34 , E1 0.0, E2 0.0, E3 0.0, E4 0.0, E5 0.0, E6 0.0}
DECL VW_MPARA_TYP P82_D = {TOOL_NO 1,BASE_NO 2,VB 200,VE 40,ACC 50,TRG_TIME 0,MOVE_TYPE #GLUE_MOTION}
DECL E6POS P82 = {X 1663.175, Y -844.2018, Z 34.56573, A -88.01324, B 17.00237, C 60.00632, S 2, T 34 , E1 0.0, E2 0.0, E3 0.0, E4 0.0, E5 0.0, E6 0.0}
DECL VW_MPARA_TYP P83_D = {TOOL_NO 1,BASE_NO 2,VB 200,VE 40,ACC 50,TRG_TIME 0,MOVE_TYPE #GLUE_MOTION}
DECL E6POS P83 = {X 1701.648, Y -843.8079, Z 36.00403, A -88.05476, B 16.97078, C 60.00671, S 2, T 34 , E1 0.0, E2 0.0, E3 0.0, E4 0.0, E5 0.0, E6 0.0}
DECL VW_MPARA_TYP P84_D = {TOOL_NO 1,BASE_NO 2,VB 200,VE 40,ACC 50,TRG_TIME 0,MOVE_TYPE #GLUE_MOTION}
DECL E6POS P84 = {X 1747.87, Y -842.947, Z 35.94467, A -88.04691, B 16.87285, C 60.02341, S 2, T 34 , E1 0.0, E2 0.0, E3 0.0, E4 0.0, E5 0.0, E6 0.0}
DECL VW_MPARA_TYP P85_D = {TOOL_NO 1,BASE_NO 2,VB 200,VE 40,ACC 50,TRG_TIME 0,MOVE_TYPE #GLUE_MOTION}
DECL E6POS P85 = {X 1758.388, Y -842.7318, Z 35.84744, A -88.03526, B 16.91858, C 60.03131, S 2, T 34 , E1 0.0, E2 0.0, E3 0.0, E4 0.0, E5 0.0, E6 0.0}
DECL VW_MPARA_TYP P86_D = {TOOL_NO 1,BASE_NO 2,VB 200,VE 40,ACC 50,TRG_TIME 0,MOVE_TYPE #GLUE_MOTION}
DECL E6POS P86 = {X 1857.363, Y -840.8391, Z 36.40408, A -87.99953, B 17.03403, C 60.1251, S 2, T 42 , E1 0.0, E2 0.0, E3 0.0, E4 0.0, E5 0.0, E6 0.0}
DECL VW_MPARA_TYP P87_D = {TOOL_NO 1,BASE_NO 2,VB 200,VE 40,ACC 50,TRG_TIME 0,MOVE_TYPE #GLUE_MOTION}
DECL E6POS P87 = {X 1894.085, Y -839.5034, Z 36.32517, A -88.01498, B 17.00514, C 60.07638, S 2, T 42 , E1 0.0, E2 0.0, E3 0.0, E4 0.0, E5 0.0, E6 0.0}
DECL VW_MPARA_TYP P88_D = {TOOL_NO 1,BASE_NO 2,VB 200,VE 40,ACC 50,TRG_TIME 0,MOVE_TYPE #GLUE_MOTION}
DECL E6POS P88 = {X 1919.268, Y -839.3327, Z 36.01661, A -88.02868, B 17.04852, C 60.01303, S 2, T 42 , E1 0.0, E2 0.0, E3 0.0, E4 0.0, E5 0.0, E6 0.0}
DECL VW_MPARA_TYP P89_D = {TOOL_NO 1,BASE_NO 2,VB 200,VE 40,ACC 50,TRG_TIME 0,MOVE_TYPE #GLUE_MOTION}
DECL E6POS P89 = {X 1941.195, Y -838.4131, Z 38.47575, A -88.0169, B 17.02987, C 60.01666, S 2, T 42 , E1 0.0, E2 0.0, E3 0.0, E4 0.0, E5 0.0, E6 0.0}
DECL VW_MPARA_TYP P90_D = {TOOL_NO 1,BASE_NO 2,VB 200,VE 40,ACC 50,TRG_TIME 0,MOVE_TYPE #GLUE_MOTION}
DECL E6POS P90 = {X 1956.498, Y -838.9611, Z 41.08417, A -87.99789, B 17.03412, C 60.00494, S 2, T 42 , E1 0.0, E2 0.0, E3 0.0, E4 0.0, E5 0.0, E6 0.0}
DECL VW_MPARA_TYP P91_D = {TOOL_NO 1,BASE_NO 2,VB 200,VE 40,ACC 50,TRG_TIME 0,MOVE_TYPE #GLUE_MOTION}
DECL E6POS P91 = {X 1966.261, Y -839.6586, Z 42.72445, A -88.01196, B 16.99745, C 59.96504, S 2, T 42 , E1 0.0, E2 0.0, E3 0.0, E4 0.0, E5 0.0, E6 0.0}
DECL VW_MPARA_TYP P92_D = {TOOL_NO 1,BASE_NO 2,VB 200,VE 40,ACC 50,TRG_TIME 0,MOVE_TYPE #GLUE_MOTION}
DECL E6POS P92 = {X 1981.502, Y -840.2649, Z 46.98776, A -87.99989, B 17.05384, C 60.04395, S 2, T 42 , E1 0.0, E2 0.0, E3 0.0, E4 0.0, E5 0.0, E6 0.0}
DECL VW_MPARA_TYP P93_D = {TOOL_NO 1,BASE_NO 2,VB 200,VE 40,ACC 50,TRG_TIME 0,MOVE_TYPE #GLUE_MOTION}
DECL E6POS P93 = {X 1995.869, Y -840.9555, Z 53.36213, A -88.14478, B 17.00766, C 60.03169, S 2, T 42 , E1 0.0, E2 0.0, E3 0.0, E4 0.0, E5 0.0, E6 0.0}
DECL VW_MPARA_TYP P94_D = {TOOL_NO 1,BASE_NO 2,VB 200,VE 40,ACC 50,TRG_TIME 0,MOVE_TYPE #GLUE_MOTION}
DECL E6POS P94 = {X 2005.013, Y -842.4586, Z 58.45709, A -88.03501, B 17.03176, C 59.97871, S 2, T 42 , E1 0.0, E2 0.0, E3 0.0, E4 0.0, E5 0.0, E6 0.0}
DECL VW_MPARA_TYP P95_D = {TOOL_NO 1,BASE_NO 2,VB 200,VE 40,ACC 50,TRG_TIME 0,MOVE_TYPE #GLUE_MOTION}
DECL E6POS P95 = {X 2014.135, Y -843.736, Z 63.13191, A -87.99748, B 17.03168, C 60.04564, S 2, T 42 , E1 0.0, E2 0.0, E3 0.0, E4 0.0, E5 0.0, E6 0.0}
DECL VW_MPARA_TYP P96_D = {TOOL_NO 1,BASE_NO 2,VB 200,VE 40,ACC 50,TRG_TIME 0,MOVE_TYPE #GLUE_MOTION}
DECL E6POS P96 = {X 2027.664, Y -844.8808, Z 71.68661, A -87.99831, B 17.01483, C 60.02847, S 2, T 42 , E1 0.0, E2 0.0, E3 0.0, E4 0.0, E5 0.0, E6 0.0}
DECL VW_MPARA_TYP P97_D = {TOOL_NO 1,BASE_NO 2,VB 200,VE 40,ACC 50,TRG_TIME 0,MOVE_TYPE #GLUE_MOTION}
DECL E6POS P97 = {X 2042.975, Y -847.3615, Z 80.824, A -88.0202, B 16.99808, C 60.02831, S 2, T 42 , E1 0.0, E2 0.0, E3 0.0, E4 0.0, E5 0.0, E6 0.0}
DECL VW_MPARA_TYP P98_D = {TOOL_NO 1,BASE_NO 2,VB 200,VE 40,ACC 50,TRG_TIME 0,MOVE_TYPE #GLUE_MOTION}
DECL E6POS P98 = {X 2059.77, Y -850.4952, Z 95.56735, A -88.06126, B 17.03467, C 59.99962, S 2, T 42 , E1 0.0, E2 0.0, E3 0.0, E4 0.0, E5 0.0, E6 0.0}
DECL VW_MPARA_TYP P99_D = {TOOL_NO 1,BASE_NO 2,VB 200,VE 40,ACC 50,TRG_TIME 0,MOVE_TYPE #GLUE_MOTION}
DECL E6POS P99 = {X 2062.937, Y -851.3162, Z 100.6355, A -88.08286, B 17.02246, C 59.99965, S 2, T 42 , E1 0.0, E2 0.0, E3 0.0, E4 0.0, E5 0.0, E6 0.0}
DECL VW_MPARA_TYP P100_D = {TOOL_NO 1,BASE_NO 2,VB 200,VE 40,ACC 50,TRG_TIME 0,MOVE_TYPE #GLUE_MOTION}
DECL E6POS P100 = {X 2064.673, Y -852.0984, Z 101.3993, A -88.05444, B 17.07561, C 60.01679, S 2, T 42 , E1 0.0, E2 0.0, E3 0.0, E4 0.0, E5 0.0, E6 0.0}
DECL VW_MPARA_TYP P101_D = {TOOL_NO 1,BASE_NO 2,VB 200,VE 40,ACC 50,TRG_TIME 0,MOVE_TYPE #GLUE_MOTION}
DECL E6POS P101 = {X 2071.878, Y -851.8516, Z 107.028, A -88.00395, B 17.02308, C 59.97105, S 2, T 42 , E1 0.0, E2 0.0, E3 0.0, E4 0.0, E5 0.0, E6 0.0}
DECL VW_MPARA_TYP P102_D = {TOOL_NO 1,BASE_NO 2,VB 200,VE 40,ACC 50,TRG_TIME 0,MOVE_TYPE #GLUE_MOTION}
DECL E6POS P102 = {X 2079.464, Y -853.093, Z 113.1263, A -88.02086, B 15.50371, C 60.04926, S 2, T 42 , E1 0.0, E2 0.0, E3 0.0, E4 0.0, E5 0.0, E6 0.0}
DECL VW_MPARA_TYP P103_D = {TOOL_NO 1,BASE_NO 2,VB 200,VE 40,ACC 50,TRG_TIME 0,MOVE_TYPE #GLUE_MOTION}
DECL E6POS P103 = {X 2083.183, Y -852.6276, Z 118.5632, A -88.1229, B 15.03134, C 60.01343, S 2, T 42 , E1 0.0, E2 0.0, E3 0.0, E4 0.0, E5 0.0, E6 0.0}
DECL VW_MPARA_TYP P104_D = {TOOL_NO 1,BASE_NO 2,VB 200,VE 40,ACC 50,TRG_TIME 0,MOVE_TYPE #GLUE_MOTION}
DECL E6POS P104 = {X 2090.684, Y -852.826, Z 126.7483, A -88.0644, B 15.03216, C 60.02255, S 2, T 42 , E1 0.0, E2 0.0, E3 0.0, E4 0.0, E5 0.0, E6 0.0}
DECL VW_MPARA_TYP P105_D = {TOOL_NO 1,BASE_NO 2,VB 200,VE 40,ACC 50,TRG_TIME 0,MOVE_TYPE #GLUE_MOTION}
DECL E6POS P105 = {X 2099.403, Y -852.0723, Z 137.6863, A -88.05429, B 14.99904, C 60.04458, S 2, T 42 , E1 0.0, E2 0.0, E3 0.0, E4 0.0, E5 0.0, E6 0.0}
DECL VW_MPARA_TYP P106_D = {TOOL_NO 1,BASE_NO 2,VB 200,VE 40,ACC 50,TRG_TIME 0,MOVE_TYPE #GLUE_MOTION}
DECL E6POS P106 = {X 2106.876, Y -852.0482, Z 148.8128, A -88.05449, B 15.03412, C 60.04726, S 2, T 42 , E1 0.0, E2 0.0, E3 0.0, E4 0.0, E5 0.0, E6 0.0}
DECL VW_MPARA_TYP P107_D = {TOOL_NO 1,BASE_NO 2,VB 200,VE 40,ACC 50,TRG_TIME 0,MOVE_TYPE #GLUE_MOTION}
DECL E6POS P107 = {X 2117.913, Y -852.494, Z 164.3103, A -88.0014, B 14.48056, C 60.01156, S 2, T 42 , E1 0.0, E2 0.0, E3 0.0, E4 0.0, E5 0.0, E6 0.0}
DECL VW_MPARA_TYP P108_D = {TOOL_NO 1,BASE_NO 2,VB 200,VE 40,ACC 50,TRG_TIME 0,MOVE_TYPE #GLUE_MOTION}
DECL E6POS P108 = {X 2128.72, Y -853.8646, Z 180.6906, A -88.16917, B 14.52523, C 60.0904, S 2, T 42 , E1 0.0, E2 0.0, E3 0.0, E4 0.0, E5 0.0, E6 0.0}
DECL VW_MPARA_TYP P109_D = {TOOL_NO 1,BASE_NO 2,VB 200,VE 40,ACC 50,TRG_TIME 0,MOVE_TYPE #GLUE_MOTION}
DECL E6POS P109 = {X 2145.225, Y -855.5547, Z 206.9787, A -88.12703, B 13.93352, C 60.04941, S 2, T 42 , E1 0.0, E2 0.0, E3 0.0, E4 0.0, E5 0.0, E6 0.0}
DECL VW_MPARA_TYP P110_D = {TOOL_NO 1,BASE_NO 2,VB 200,VE 40,ACC 50,TRG_TIME 0,MOVE_TYPE #GLUE_MOTION}
DECL E6POS P110 = {X 2168.094, Y -857.3237, Z 241.5721, A -88.04613, B 13.06301, C 60.02808, S 2, T 42 , E1 0.0, E2 0.0, E3 0.0, E4 0.0, E5 0.0, E6 0.0}
DECL VW_MPARA_TYP P111_D = {TOOL_NO 1,BASE_NO 2,VB 200,VE 40,ACC 50,TRG_TIME 0,MOVE_TYPE #GLUE_MOTION}
DECL E6POS P111 = {X 2218.219, Y -859.4075, Z 312.7245, A -88.01942, B 12.3937, C 60.02275, S 2, T 42 , E1 0.0, E2 0.0, E3 0.0, E4 0.0, E5 0.0, E6 0.0}
DECL VW_MPARA_TYP P112_D = {TOOL_NO 1,BASE_NO 2,VB 200,VE 40,ACC 50,TRG_TIME 0,MOVE_TYPE #GLUE_MOTION}
DECL E6POS P112 = {X 2234.939, Y -860.5358, Z 340.6331, A -88.01091, B 12.29758, C 60.12138, S 2, T 42 , E1 0.0, E2 0.0, E3 0.0, E4 0.0, E5 0.0, E6 0.0}
DECL VW_MPARA_TYP P113_D = {TOOL_NO 1,BASE_NO 2,VB 200,VE 40,ACC 50,TRG_TIME 0,MOVE_TYPE #GLUE_MOTION}
DECL E6POS P113 = {X 2253.58, Y -862.1984, Z 369.7937, A -88.02818, B 11.94102, C 59.98626, S 2, T 42 , E1 0.0, E2 0.0, E3 0.0, E4 0.0, E5 0.0, E6 0.0}
DECL VW_MPARA_TYP P114_D = {TOOL_NO 1,BASE_NO 2,VB 200,VE 40,ACC 50,TRG_TIME 0,MOVE_TYPE #GLUE_MOTION}
DECL E6POS P114 = {X 2262.456, Y -861.5928, Z 383.922, A -87.98428, B 11.8582, C 60.00203, S 2, T 42 , E1 0.0, E2 0.0, E3 0.0, E4 0.0, E5 0.0, E6 0.0}
DECL VW_MPARA_TYP P115_D = {TOOL_NO 1,BASE_NO 2,VB 200,VE 40,ACC 50,TRG_TIME 0,MOVE_TYPE #GLUE_MOTION}
DECL E6POS P115 = {X 2276.468, Y -861.7311, Z 409.4049, A -87.91366, B 11.49988, C 60.13818, S 2, T 42 , E1 0.0, E2 0.0, E3 0.0, E4 0.0, E5 0.0, E6 0.0}
DECL VW_MPARA_TYP P116_D = {TOOL_NO 1,BASE_NO 2,VB 200,VE 40,ACC 50,TRG_TIME 0,MOVE_TYPE #GLUE_MOTION}
DECL E6POS P116 = {X 2288.736, Y -860.631, Z 430.3949, A -87.95031, B 10.95198, C 60.03755, S 2, T 42 , E1 0.0, E2 0.0, E3 0.0, E4 0.0, E5 0.0, E6 0.0}
DECL VW_MPARA_TYP P117_D = {TOOL_NO 1,BASE_NO 2,VB 200,VE 40,ACC 50,TRG_TIME 0,MOVE_TYPE #GLUE_MOTION}
DECL E6POS P117 = {X 2295.188, Y -860.2522, Z 440.7064, A -88.05811, B 10.90242, C 60.05781, S 2, T 42 , E1 0.0, E2 0.0, E3 0.0, E4 0.0, E5 0.0, E6 0.0}
DECL VW_MPARA_TYP P118_D = {TOOL_NO 1,BASE_NO 2,VB 200,VE 40,ACC 50,TRG_TIME 0,MOVE_TYPE #GLUE_MOTION}
DECL E6POS P118 = {X 2304.61, Y -859.4771, Z 454.6766, A -88.04729, B 10.74358, C 60.08749, S 2, T 42 , E1 0.0, E2 0.0, E3 0.0, E4 0.0, E5 0.0, E6 0.0}
DECL VW_MPARA_TYP P119_D = {TOOL_NO 1,BASE_NO 2,VB 200,VE 40,ACC 50,TRG_TIME 0,MOVE_TYPE #GLUE_MOTION}
DECL E6POS P119 = {X 2312.589, Y -858.3376, Z 467.3503, A -87.73141, B 10.68322, C 60.06334, S 2, T 42 , E1 0.0, E2 0.0, E3 0.0, E4 0.0, E5 0.0, E6 0.0}
DECL VW_MPARA_TYP P120_D = {TOOL_NO 1,BASE_NO 2,VB 200,VE 40,ACC 50,TRG_TIME 0,MOVE_TYPE #GLUE_MOTION}
DECL E6POS P120 = {X 2333.329, Y -852.8982, Z 493.3136, A -88.03075, B 9.857472, C 59.94152, S 2, T 42 , E1 0.0, E2 0.0, E3 0.0, E4 0.0, E5 0.0, E6 0.0}
DECL VW_MPARA_TYP P121_D = {TOOL_NO 1,BASE_NO 2,VB 200,VE 40,ACC 50,TRG_TIME 0,MOVE_TYPE #GLUE_MOTION}
DECL E6POS P121 = {X 2358.241, Y -842.1559, Z 536.761, A -88.14795, B 9.236975, C 60.19158, S 2, T 42 , E1 0.0, E2 0.0, E3 0.0, E4 0.0, E5 0.0, E6 0.0}
DECL VW_MPARA_TYP P122_D = {TOOL_NO 1,BASE_NO 2,VB 200,VE 40,ACC 50,TRG_TIME 0,MOVE_TYPE #GLUE_MOTION}
DECL E6POS P122 = {X 2367.959, Y -835.8517, Z 553.7233, A -88.11703, B 8.30783, C 60.13571, S 2, T 42 , E1 0.0, E2 0.0, E3 0.0, E4 0.0, E5 0.0, E6 0.0}
DECL VW_MPARA_TYP P123_D = {TOOL_NO 1,BASE_NO 2,VB 200,VE 40,ACC 50,TRG_TIME 0,MOVE_TYPE #GLUE_MOTION}
DECL E6POS P123 = {X 2379.917, Y -829.5908, Z 570.2271, A -88.08709, B 7.40379, C 60.08085, S 2, T 42 , E1 0.0, E2 0.0, E3 0.0, E4 0.0, E5 0.0, E6 0.0}
DECL VW_MPARA_TYP P124_D = {TOOL_NO 1,BASE_NO 2,VB 200,VE 40,ACC 50,TRG_TIME 0,MOVE_TYPE #GLUE_MOTION}
DECL E6POS P124 = {X 2389.097, Y -824.1639, Z 584.5319, A -88.06124, B 6.620198, C 60.03291, S 2, T 42 , E1 0.0, E2 0.0, E3 0.0, E4 0.0, E5 0.0, E6 0.0}
DECL VW_MPARA_TYP P125_D = {TOOL_NO 1,BASE_NO 2,VB 200,VE 40,ACC 50,TRG_TIME 0,MOVE_TYPE #GLUE_MOTION}
DECL E6POS P125 = {X 2410.635, Y -813.9879, Z 610.6584, A -88.01333, B 5.161689, C 59.94272, S 2, T 42 , E1 0.0, E2 0.0, E3 0.0, E4 0.0, E5 0.0, E6 0.0}
DECL VW_MPARA_TYP P126_D = {TOOL_NO 1,BASE_NO 2,VB 200,VE 40,ACC 50,TRG_TIME 0,MOVE_TYPE #GLUE_MOTION}
DECL E6POS P126 = {X 2416.476, Y -809.3995, Z 620.2584, A -88.06689, B 4.671606, C 59.9285, S 2, T 42 , E1 0.0, E2 0.0, E3 0.0, E4 0.0, E5 0.0, E6 0.0}
DECL VW_MPARA_TYP P127_D = {TOOL_NO 1,BASE_NO 2,VB 200,VE 40,ACC 50,TRG_TIME 0,MOVE_TYPE #GLUE_MOTION}
DECL E6POS P127 = {X 2423.009, Y -807.0663, Z 628.3654, A -88.11546, B 4.226681, C 59.91599, S 2, T 42 , E1 0.0, E2 0.0, E3 0.0, E4 0.0, E5 0.0, E6 0.0}
DECL VW_MPARA_TYP P128_D = {TOOL_NO 1,BASE_NO 2,VB 200,VE 40,ACC 50,TRG_TIME 0,MOVE_TYPE #GLUE_MOTION}
DECL E6POS P128 = {X 2432.363, Y -804.4048, Z 637.7181, A -88.07281, B 3.558602, C 59.87203, S 2, T 42 , E1 0.0, E2 0.0, E3 0.0, E4 0.0, E5 0.0, E6 0.0}
DECL VW_MPARA_TYP P129_D = {TOOL_NO 1,BASE_NO 2,VB 200,VE 40,ACC 50,TRG_TIME 0,MOVE_TYPE #GLUE_MOTION}
DECL E6POS P129 = {X 2433.688, Y -799.4921, Z 645.8392, A -88.0377, B 3.007927, C 59.83541, S 2, T 42 , E1 0.0, E2 0.0, E3 0.0, E4 0.0, E5 0.0, E6 0.0}
DECL VW_MPARA_TYP P130_D = {TOOL_NO 1,BASE_NO 2,VB 200,VE 40,ACC 50,TRG_TIME 0,MOVE_TYPE #GLUE_MOTION}
DECL E6POS P130 = {X 2439.84, Y -786.485, Z 658.6435, A -88.03258, B 2.045004, C 59.73536, S 2, T 42 , E1 0.0, E2 0.0, E3 0.0, E4 0.0, E5 0.0, E6 0.0}
DECL VW_MPARA_TYP P131_D = {TOOL_NO 1,BASE_NO 2,VB 200,VE 40,ACC 50,TRG_TIME 0,MOVE_TYPE #GLUE_MOTION}
DECL E6POS P131 = {X 2443.815, Y -777.5999, Z 667.2053, A -88.02899, B 1.370112, C 59.66518, S 2, T 42 , E1 0.0, E2 0.0, E3 0.0, E4 0.0, E5 0.0, E6 0.0}
DECL VW_MPARA_TYP P132_D = {TOOL_NO 1,BASE_NO 2,VB 200,VE 40,ACC 50,TRG_TIME 0,MOVE_TYPE #GLUE_MOTION}
DECL E6POS P132 = {X 2452.246, Y -766.5745, Z 677.8301, A -88.02435, B 0.4963125, C 59.57426, S 2, T 42 , E1 0.0, E2 0.0, E3 0.0, E4 0.0, E5 0.0, E6 0.0}
DECL VW_MPARA_TYP P133_D = {TOOL_NO 1,BASE_NO 2,VB 200,VE 40,ACC 50,TRG_TIME 0,MOVE_TYPE #GLUE_MOTION}
DECL E6POS P133 = {X 2461.837, Y -753.591, Z 692.3879, A -88.01829, B -0.6466179, C 59.45522, S 2, T 42 , E1 0.0, E2 0.0, E3 0.0, E4 0.0, E5 0.0, E6 0.0}
DECL VW_MPARA_TYP P134_D = {TOOL_NO 1,BASE_NO 2,VB 200,VE 40,ACC 50,TRG_TIME 0,MOVE_TYPE #GLUE_MOTION}
DECL E6POS P134 = {X 2470.04, Y -740.9911, Z 708.9511, A -88.0116, B -1.90697, C 59.32382, S 2, T 42 , E1 0.0, E2 0.0, E3 0.0, E4 0.0, E5 0.0, E6 0.0}
DECL VW_MPARA_TYP P135_D = {TOOL_NO 1,BASE_NO 2,VB 200,VE 40,ACC 50,TRG_TIME 0,MOVE_TYPE #GLUE_MOTION}
DECL E6POS P135 = {X 2475.97, Y -732.4688, Z 721.2266, A -88.00648, B -2.870632, C 59.22325, S 2, T 42 , E1 0.0, E2 0.0, E3 0.0, E4 0.0, E5 0.0, E6 0.0}
DECL VW_MPARA_TYP P136_D = {TOOL_NO 1,BASE_NO 2,VB 200,VE 40,ACC 50,TRG_TIME 0,MOVE_TYPE #GLUE_MOTION}
DECL E6POS P136 = {X 2482.0, Y -725.0536, Z 731.9072, A -88.00201, B -3.709092, C 59.13567, S 2, T 42 , E1 0.0, E2 0.0, E3 0.0, E4 0.0, E5 0.0, E6 0.0}
DECL VW_MPARA_TYP P137_D = {TOOL_NO 1,BASE_NO 2,VB 200,VE 10,ACC 50,TRG_TIME 5,MOVE_TYPE #GLUE_MOTION}
DECL E6POS P137 = {X 2489.991, Y -720.2316, Z 739.6482, A -88.01206, B -6.349968, C 58.48532, S 2, T 34 , E1 0.0, E2 0.0, E3 0.0, E4 0.0, E5 0.0, E6 0.0}
DECL VW_MPARA_TYP P138_D = {TOOL_NO 1,BASE_NO 2,VB 200,VE 40,ACC 50,TRG_TIME 0,MOVE_TYPE #GLUE_MOTION}
DECL E6POS P138 = {X 2489.991, Y -687.1135, Z 739.696, A -88.01206, B -6.349968, C 58.48532, S 2, T 34 , E1 0.0, E2 0.0, E3 0.0, E4 0.0, E5 0.0, E6 0.0}
DECL VW_MPARA_TYP P139_D = {TOOL_NO 1,BASE_NO 2,VB 100,VE 100,ACC 100,TRG_TIME 0,MOVE_TYPE #PTP_MOTION}
DECL E6POS P139 = {X 2449.527, Y -683.7665, Z 730.7533, A -88.02371, B -1.352956, C 58.6586, S 2, T 42 , E1 0.0, E2 0.0, E3 0.0, E4 0.0, E5 0.0, E6 0.0}
DECL VW_MPARA_TYP P140_D = {TOOL_NO 1,BASE_NO 2,VB 100,VE 100,ACC 100,TRG_TIME 0,MOVE_TYPE #PTP_MOTION}
DECL E6POS P140 = {X 2491.435, Y -588.4056, Z 786.3615, A -88.12092, B -19.55178, C 25.00472, S 2, T 34 , E1 0.0, E2 0.0, E3 0.0, E4 0.0, E5 0.0, E6 0.0}
DECL VW_MPARA_TYP P141_D = {TOOL_NO 1,BASE_NO 2,VB 100,VE 100,ACC 100,TRG_TIME 0,MOVE_TYPE #PTP_MOTION}
DECL E6POS P141 = {X 2944.878, Y 763.7927, Z 360.1338, A -39.35303, B -11.92739, C -28.43664, S 2, T 42 , E1 0.0, E2 0.0, E3 0.0, E4 0.0, E5 0.0, E6 0.0}
DECL VW_MPARA_TYP P142_D = {TOOL_NO 1,BASE_NO 2,VB 100,VE 100,ACC 100,TRG_TIME 0,MOVE_TYPE #PTP_MOTION}
DECL E6POS P142 = {X 2338.384, Y 800.6096, Z -2898.13, A -131.9922, B 48.17278, C -165.2234, S 2, T 43 , E1 0.0, E2 0.0, E3 0.0, E4 0.0, E5 0.0, E6 0.0}
DECL VW_MPARA_TYP P143_D = {TOOL_NO 1,BASE_NO 2,VB 100,VE 100,ACC 100,TRG_TIME 0,MOVE_TYPE #PTP_MOTION}
DECL E6POS P143 = {X 2277.056, Y -421.1326, Z -1906.485, A -89.9705, B -0.0342025, C 61.11638, S 2, T 3 , E1 0.0, E2 0.0, E3 0.0, E4 0.0, E5 0.0, E6 0.0}
DECL VW_MPARA_TYP P144_D = {TOOL_NO 1,BASE_NO 2,VB 100,VE 0,ACC 100,TRG_TIME 0,MOVE_TYPE #PTP_MOTION}
DECL E6POS P144 = {X 2277.11, Y -526.3644, Z -1906.422, A -89.9705, B -0.03420252, C 61.11638, S 2, T 3 , E1 0.0, E2 0.0, E3 0.0, E4 0.0, E5 0.0, E6 0.0}
ENDDAT
